    arCamPoint_4p[3].FunctionType := MOTIONFUNCTYPE_BESCHLTRAPEZ_VR;
    arCamPoint_4p[3].MasterPos    := Curve3_MasterPosition;
    arCamPoint_4p[3].SlavePos     := Curve3_SlavePosition;
    arCamPoint_4p[3].PointIndex   := 4;
    arCamPoint_4p[3].PointType    := MOTIONPOINTTYPE_REST;

    arCamPoint_4p[4].FunctionType := MOTIONFUNCTYPE_POLYNOM1;
    arCamPoint_4p[4].MasterPos    := Curve4_MasterPosition;
    arCamPoint_4p[4].SlavePos     := Curve4_SlavePosition;
    arCamPoint_4p[4].PointIndex   := 5;
    arCamPoint_4p[4].PointType    := MOTIONPOINTTYPE_REST;

END_IF
END_METHOD

METHOD StartAction
VAR_OUTPUT
    xComplete : BOOL := TRUE;
	iErrorID : INT := 0;
END_VAR
// Check Parameter is correct
// Data analyze
WheelThreadCircumference := WheelThreadDiameter * PI;                          // (mm)
PrintCircumference       := PrintRollerDiameter * PI;                          // (mm)
MaxMachineLineSpeed      := PrintRollerDiameter * PI * MaxMasterVelocity / 60; // (mm/s)
MachineLineSpeed         := PrintCircumference * MasterVelocity / 60;          // (mm/s)

SlaveLineSpeedScale := (PrintRollerDiameter / WheelThreadDiameter) * 360 / 60; // (deg/s)

MaxSlaveLineSpeed := SlaveLineSpeedScale * MaxMasterVelocity; // (deg/s)

SlaveSyncSpeed        := SlaveLineSpeedScale * MasterVelocity;              // (deg/s)
SlaveSyncDistance     := ProductLength - AccDistance - WheelThreadPosition; // (mm)
SlaveSyncDistance_deg := (SlaveSyncDistance / WheelThreadCircumference) * 360;

SlaveSyncTime     := SlaveSyncDistance_Deg / SlaveSyncSpeed; // (sec)
SlaveSyncTime_deg := (SlaveSyncTime / 60 * MasterVelocity) * 360;
SlaveWaitGapTime  := (GapOfProduct / PrintCircumference) * 360 / SlaveSyncSpeed; // (sec)
GapOfProduct_deg  := (SlaveWaitGapTime / 60 * MasterVelocity) * 360;
AccTime           := SQRT(AccDistance / ((MaxAcceleration * 0.5) - (MaxAcceleration / 3) + (MaxAcceleration / 4)));
AccTime_deg       := (AccTime / 60 * MasterVelocity) * 360;
AccDistance_deg   := (AccDistance / WheelThreadCircumference) * 360;
//(Sf := AccDistance, Tout => MasterAccDeg);
MasterAccDeg := F_Poly7_MinTime(EndPosition := AccDistance, EndVelocity := MachineLineSpeed);
// Data input 
Curve1_MasterPosition := 5 * MasterAccDeg;
Curve1_SlavePosition  := AccDistance;
Curve2_MasterPosition := 5 * MasterAccDeg + SlaveSyncTime_deg;
Curve2_SlavePosition  := AccDistance + SlaveSyncDistance;

IF ((360 - Curve2_MasterPosition) > 21.5) OR ((ProductLength - Curve2_SlavePosition) > 50) THEN
    Curve4_active         := TRUE;
	IF ((360 - Curve2_MasterPosition) > 21.5) THEN
    	Curve3_MasterPosition := Curve2_MasterPosition + 21.5;
	ELSE
		Curve3_MasterPosition := Curve2_MasterPosition;
	END_IF
	IF ((ProductLength - Curve2_SlavePosition) > 50) THEN
    	Curve3_SlavePosition  := Curve2_SlavePosition +50;
	ELSE	
		Curve3_SlavePosition := ProductLength;
	END_IF
	Curve4_MasterPosition := 360;
	Curve4_SlavePosition := ProductLength;
ELSE
    Curve4_active         := FALSE;
    Curve3_MasterPosition := 360;
    Curve3_SlavePosition  := ProductLength;
END_IF
END_METHOD

END_FUNCTION_BLOCK

// Main
PROGRAM Main 
VAR
	bJogP: BOOL;
	bJogN: BOOL;
	rVelocityCmd: LREAL;
	bPTP : BOOL;
	bSyncVel : BOOL;
	rPosAbsCmd: LREAL;
	bSetPosition : BOOL;
	bSyncPhase : BOOL;
	bSyncProfile:BOOL;
	//fbCalculateFeederCurve : FB_CorrugatedWheelThread;
	fbWheelThreadCal : FB_CorrugatedWheelThreadCalculate;
	fbLiftingCal : FB_CorrugatedLiftingCalculate;
//	MasterAccDeg : LREAL;
	bHoming		:BOOL;
	bPTP_Execute : BOOL;
	bEstop: BOOL := TRUE;
	bModeAH : BOOL;
	MasterSyncPos : LREAL;
	SlaveSyncPos : LREAL;
	bPhaseAbs_Execute :BOOL;
	bSyncVel_Test: BOOL;
	AniloxLowSpeed : LREAL:=10;
	bSyncPhase_Test : BOOL;
END_VAR

// Implement AxisInterface
AxisInterface_Type01();

//fbCalculateFeederCurve();
IF NOT bJogN AND_THEN bJogP THEN
	arAxisCtrl_gb[1].VelMode.Acc      := 100;
	arAxisCtrl_gb[1].VelMode.Dec      := 100;
	arAxisCtrl_gb[1].VelMode.Jerk     := 1000;
	arAxisCtrl_gb[1].VelMode.Velocity := rVelocityCmd;
	arAxisCtrl_gb[1].Admin._OpMode.en := ModeVel;

ELSIF NOT bJogP AND_THEN bJogN THEN
	arAxisCtrl_gb[1].VelMode.Acc      := 100;
	arAxisCtrl_gb[1].VelMode.Dec      := 100;
	arAxisCtrl_gb[1].VelMode.Jerk     := 1000;
	arAxisCtrl_gb[1].VelMode.Velocity := -rVelocityCmd;
	arAxisCtrl_gb[1].Admin._OpMode.en := ModeVel;
ELSIF bPTP THEN
	arAxisCtrl_gb[1].PosMode.Acc      := 100;
	arAxisCtrl_gb[1].PosMode.Dec      := 100;
	arAxisCtrl_gb[1].PosMode.Jerk     := 1000;
	arAxisCtrl_gb[1].PosMode.Velocity := rVelocityCmd;
	arAxisCtrl_gb[1].PosMode.Position := rPosAbsCmd;
	arAxisCtrl_gb[1].Admin._OpMode.en := ModePosAbs;
ELSIF bSetPosition THEN
	(*arAxisCtrl_gb[1].SetupMode.SetPosition_Position := rPosAbsCmd;
	arAxisCtrl_gb[1].SetupMode.HomingMode := E_HomingMode.CurrentPosition;
	arAxisCtrl_gb[1].Admin._OpMode.en := ModeHoming;*)
ELSIF bHoming THEN

	arAxisCtrl_gb[1].SetupMode.FastVelo.Velocity := 1000;
	arAxisCtrl_gb[1].SetupMode.FastVelo.Acc      := 10000;
	arAxisCtrl_gb[1].SetupMode.FastVelo.Dec      := 10000;
	arAxisCtrl_gb[1].SetupMode.FastVelo.Jerk     := 100000;

	arAxisCtrl_gb[1].SetupMode.SlowVelo.Velocity := 1;
	arAxisCtrl_gb[1].SetupMode.SlowVelo.Acc      := 10;
	arAxisCtrl_gb[1].SetupMode.SlowVelo.Dec      := 10;
	arAxisCtrl_gb[1].SetupMode.SlowVelo.Jerk     := 100;

	arAxisCtrl_gb[1].Admin._OpMode.en := ModeHoming;

ELSIF bModeAH THEN
	arAxisCtrl_gb[1].Admin._OpMode.en := ModeAH;
ELSE
	arAxisCtrl_gb[1].Admin._OpMode.en := ModeAb;
END_IF
arAxisCtrl_gb[1].Admin._OpMode.b.ModeStopping := NOT bEstop;

IF bSyncVel THEN
	arAxisCtrl_gb[2].SyncMode.SyncVel.Acceleration     := 10000;
	arAxisCtrl_gb[2].SyncMode.SyncVel.Deceleration     := 10000;
	arAxisCtrl_gb[2].SyncMode.SyncVel.Jerk             := 100000;
	arAxisCtrl_gb[2].SyncMode.SyncVel.FineAdjust       := 0;
	arAxisCtrl_gb[2].SyncMode.SyncVel.InputRevolution  := 1;
	arAxisCtrl_gb[2].SyncMode.SyncVel.OutputRevolution := 1;
	arAxisCtrl_gb[2].SyncMode.SyncVel.Master           := (arAxisCtrl_gb[1].Admin.Axis);
	arAxisCtrl_gb[2].Admin._OpMode.en                  := ModeSyncVel;
ELSIF bSyncPhase THEN
	arAxisCtrl_gb[2].SyncMode.SyncPhase.MaxAcceleration  := 10000;
	arAxisCtrl_gb[2].SyncMode.SyncPhase.MaxDeceleration  := 10000;
	arAxisCtrl_gb[2].SyncMode.SyncPhase.MaxJerk          := 100000;
	arAxisCtrl_gb[2].SyncMode.SyncPhase.InputRevolution  := 1;
	arAxisCtrl_gb[2].SyncMode.SyncPhase.OutputRevolution := 1;
	arAxisCtrl_gb[2].SyncMode.SyncPhase.MaxVelocity      := 1000;
	arAxisCtrl_gb[2].SyncMode.SyncPhase.MasterSyncPos    := MasterSyncPos;
	arAxisCtrl_gb[2].SyncMode.SyncPhase.SlaveSyncPos     := SlaveSyncPos;
	arAxisCtrl_gb[2].SyncMode.SyncPhase.SyncVelocity := 60;
	arAxisCtrl_gb[2].SyncMode.SyncPhase.SyncAcceleration := 1000;
	arAxisCtrl_gb[2].SyncMode.SyncPhase.Master           := arAxisCtrl_gb[1].Admin.Axis;
	arAxisCtrl_gb[2].Admin.PositionType                  := E_PositionType.Modulo;
	arAxisCtrl_gb[2].Admin._OpMode.en                    := ModeSyncPhase;
ELSIF bSyncProfile THEN
	arAxisCtrl_gb[2].SyncMode.SyncProfile.MasterAxis := arAxisCtrl_gb[1].Admin.Axis;
	arAxisCtrl_gb[2].SyncMode.SyncProfile.Periodic   := TRUE;
	arAxisCtrl_gb[2].SyncMode.SyncProfile.ProfileNum := 1;
	arAxisCtrl_gb[2].SyncMode.SyncProfile.SyncType   := MC_StartMode.MC_STARTMODE_RELATIVE;
	arAxisCtrl_gb[2].Admin._OpMode.en                := ModeSyncProfile;
ELSIF bPTP_Execute THEN
	arAxisCtrl_gb[1].PosMode.Acc      := 100;
	arAxisCtrl_gb[1].PosMode.Dec      := 100;
	arAxisCtrl_gb[1].PosMode.Jerk     := 1000;
	arAxisCtrl_gb[1].PosMode.Position := 20;
	arAxisCtrl_gb[1].PosMode.Velocity := 2;
ELSIF bSyncVel_Test THEN
	IF arAxisCtrl_gb[1].Admin.Axis.NcToPlc.ActVelo >= 10 THEN
//		arAxisCtrl_gb[2].SyncMode.SyncPhase.MaxAcceleration  := 10000;
//		arAxisCtrl_gb[2].SyncMode.SyncPhase.MaxDeceleration  := 10000;
//		arAxisCtrl_gb[2].SyncMode.SyncPhase.MaxJerk          := 100000;
//		arAxisCtrl_gb[2].SyncMode.SyncPhase.InputRevolution  := 1;
//		arAxisCtrl_gb[2].SyncMode.SyncPhase.OutputRevolution := 1;
//		arAxisCtrl_gb[2].SyncMode.SyncPhase.MaxVelocity      := 1000;
//		arAxisCtrl_gb[2].SyncMode.SyncPhase.MasterSyncPos    := MasterSyncPos;
//		arAxisCtrl_gb[2].SyncMode.SyncPhase.SlaveSyncPos     := SlaveSyncPos;
//		arAxisCtrl_gb[2].SyncMode.SyncPhase.Master           := arAxisCtrl_gb[1].Admin.Axis;
//		arAxisCtrl_gb[2].Admin.PositionType                  := E_PositionType.Modulo;
//		arAxisCtrl_gb[2].Admin._OpMode.en                    := ModeSyncPhase;
	ELSIF arAxisCtrl_gb[1].Admin.Axis.NcToPlc.ActVelo < 10 THEN
		arAxisCtrl_gb[2].VelMode.Acc      := 100;
		arAxisCtrl_gb[2].VelMode.Dec      := 100;
		arAxisCtrl_gb[2].VelMode.Jerk     := 1000;
		arAxisCtrl_gb[2].VelMode.Velocity := AniloxLowSpeed;
		arAxisCtrl_gb[2].Admin._OpMode.en := E_AXIS_MODE.ModeVel;

	END_IF
ELSIF bSyncPhase_Test THEN
	arAxisCtrl_gb[2].Admin.PositionType := E_PositionType.Modulo;
	arAxisCtrl_gb[2].SyncMode.SyncPhase.Master := arAxisCtrl_gb[1].Admin.Axis;
	arAxisCtrl_gb[2].SyncMode.SyncPhase.InputRevolution := 1;
	arAxisCtrl_gb[2].SyncMode.SyncPhase.OutputRevolution :=1;
//	arAxisCtrl_gb[2].SyncMode.SyncPhase.PhaseOffsetVel := 10;
//	arAxisCtrl_gb[2].SyncMode.SyncPhase.PhaseOffsetAcc := 100;
//	arAxisCtrl_gb[2].SyncMode.SyncPhase.StartMode := E_StartMode.Absolute;
//	arAxisCtrl_gb[2].SyncMode.SyncPhase.SyncVelocity := 10;
//	arAxisCtrl_gb[2].SyncMode.SyncPhase.SyncAcceleration := 100;

	arAxisCtrl_gb[2].SyncMode.SyncPhase.Master := arAxisCtrl_gb[1].Admin.Axis;
	arAxisCtrl_gb[2].SyncMode.SyncPhase.InputRevolution := 1;
	arAxisCtrl_gb[2].SyncMode.SyncPhase.OutputRevolution := 1;
	arAxisCtrl_gb[2].SyncMode.SyncPhase.MaxVelocity := 2000;
	arAxisCtrl_gb[2].SyncMode.SyncPhase.MaxAcceleration := 1500;
	arAxisCtrl_gb[2].SyncMode.SyncPhase.MaxDeceleration := 1500;
	arAxisCtrl_gb[2].SyncMode.SyncPhase.MaxJerk := 2250;
	



	arAxisCtrl_gb[2].Admin._OpMode.en := E_AXIS_MODE.ModeSyncPhase;
ELSE
	arAxisCtrl_gb[2].Admin._OpMode.en := ModeAH;
END_IF


fbWheelThreadCal(xDone =>,
                 xBusy =>,
                 xError =>,
                 xExecute :=,
                 xAbort :=,
                 ProfileNum := 1,
                 MaxMasterVelocity :=,
                 ProductLength := 1300,
                 AccDistance :=,
                 WheelThreadPosition :=,
                 WheelThreadDiameter :=,
                 PrintRollerDiameter :=,
                 MasterVelocity :=,
                 GapOfProduct :=,
                 MaxAcceleration :=,
                 AxisID := 2,
                 xAborted =>);
fbLiftingCal(xDone =>,
             xBusy =>,
             xError =>,
             xExecute :=,
             xAbort :=,
             AxisID := 2,
             ProfileNum := 1,
             WorkingAreaStartPos :=,
             WorkingAreaEndPos :=,
             MaxMasterVelocity :=,
             ProductLength := 1300,
             PrintRollerDiameter :=,
             SlaveWorkLength :=,
             WheelThreadPosition :=,
             xAborted =>);

END_PROGRAM
